FUNCTION_BLOCK FB_TwoAxisPopIn
VAR_INPUT
	RepRate : BOOL;
	
	Axis1_InsertedPos2_IN : BOOL;
	Axis1_RetractedPos1_IN : BOOL;
	
	Axis2_InsertedPos2_IN : BOOL;
	Axis2_RetractedPos1_IN : BOOL;
END_VAR
VAR_OUTPUT
	Interlock : BOOL;
	Axis1_State : E_2PosMonState;
	Axis2_State : E_2PosMonState;
	
	Axis1_InsertPos2_OUT : BOOL;
	Axis2_InsertPos2_OUT : BOOL;
END_VAR
VAR
	Axis1 : FB_TwoPositionPopIn;
	Axis2 : FB_TwoPositionPopIn;
END_VAR

// Instances of 2 and 3 position monitor
Axis1(RepRate := RepRate, 	
			Inserted_Pos2_IN := Axis1_InsertedPos2_IN,	
			Retracted_Pos1_IN := Axis1_RetractedPos1_IN,
			Insert_Pos2_OUT => Axis1_InsertPos2_OUT,
			State => Axis1_State );
			
Axis2(RepRate := RepRate,  
		Inserted_Pos2_IN := Axis2_InsertedPos2_IN, 	
		Retracted_Pos1_IN := Axis2_RetractedPos1_IN,
		Insert_Pos2_OUT => Axis2_InsertPos2_OUT, 
		State => Axis2_State);

//Handle Horizontal -  RET Air solenoid - three way position monitor collisions

IF Axis1.State = E_2PosMonState.isBROKEN AND Axis2.State= E_2PosMonState.isINSERTED THEN 
	Axis1.Retract();
ELSIF Axis1.State = E_2PosMonState.isRETRACTED AND Axis2.State = E_2PosMonState.isBROKEN THEN 
	Axis1.Retract();
ELSIF Axis1.State = E_2PosMonState.isRETRACTED AND Axis2.State = E_2PosMonState.isINSERTED THEN 
	Axis1.Retract();
ELSIF Axis1.State = E_2PosMonState.isRETRACTED AND Axis2.State = E_2PosMonState.isMOVING THEN 
	Axis1.Retract();
ELSIF Axis1.State = E_2PosMonState.isMOVING AND Axis2.State = E_2PosMonState.isINSERTED THEN 
	Axis1.Retract();
ELSIF Axis1.State = E_2PosMonState.isMOVING AND Axis2.State = E_2PosMonState.isBROKEN THEN 
	Axis1.Retract();
END_IF
			
//Handle vertical 		two way position monitor collisions	
IF Axis1.State = E_2PosMonState.isBROKEN AND Axis2.State = E_2PosMonState.isRETRACTED THEN 
	Axis2.Retract();
ELSIF Axis1.State = E_2PosMonState.isBROKEN AND Axis2.State = E_2PosMonState.isMOVING THEN 
	Axis2.Retract();
ELSIF Axis1.State = E_2PosMonState.isINSERTED AND Axis2.State = E_2PosMonState.isBROKEN THEN 
	Axis2.Retract();
ELSIF Axis1.State = E_2PosMonState.isINSERTED AND Axis2.State = E_2PosMonState.isRETRACTED THEN 
	Axis2.Retract();
ELSIF Axis1.State = E_2PosMonState.isINSERTED AND Axis2.State = E_2PosMonState.isMOVING THEN 
	Axis2.Retract();
ELSIF Axis1.State = E_2PosMonState.isMOVING AND Axis2.State = E_2PosMonState.isRETRACTED THEN 
	Axis2.Retract();
END_IF

// Handle MPS shutter Interlock output
Interlock := Axis2.Interlock AND Axis1.Interlock AND 
			(Axis1.State = E_2PosMonState.isRETRACTED AND Axis2.State = E_2PosMonState.isINSERTED) OR
			(Axis1.State = E_2PosMonState.isRETRACTED AND Axis2.State = E_2PosMonState.isRETRACTED) OR
			(Axis1.State = E_2PosMonState.isINSERTED AND Axis2.State= E_2PosMonState.isRETRACTED);

METHOD Control : BOOL
VAR_IN_OUT
	structure : ST_TwoAxisPopIn;
END_VAR
//Commands
IF structure.Axis1_InsertPos2Cmd THEN
	structure.Axis1_InsertPos2Cmd:=FALSE;
	InsertAxis1();
END_IF

IF structure.Axis1_RetractPos1Cmd THEN
	structure.Axis1_RetractPos1Cmd:=FALSE;
	RetractAxis1();
END_IF

IF structure.Axis2_InsertPos2Cmd THEN
	structure.Axis2_InsertPos2Cmd:=FALSE;
	InsertAxis2();
END_IF

IF structure.Axis2_RetractPos1Cmd THEN
	structure.Axis2_RetractPos1Cmd:=FALSE;
	RetractAxis2();
END_IF

//Statuses

structure.Axis1_IsInsertedPos2St:=Axis1.Inserted_Pos2_IN;
structure.Axis1_IsRetractedPos1St:=Axis1.Retracted_Pos1_IN;

structure.Axis2_IsInsertedPos2St:=Axis2.Inserted_Pos2_IN;
structure.Axis2_IsRetractedPos1St:=Axis2.Retracted_Pos1_IN;

structure.InterlockSt:=Interlock;

structure.Axis1StateSt:=Axis1_State;
structure.Axis2StateSt:=Axis2_State;
END_METHOD

METHOD InsertAxis1 : BOOL
VAR_INPUT
END_VAR
IF Axis1.State = E_3PosMonState.isBROKEN AND Axis2.State= E_2PosMonState.isINSERTED THEN 
	RETURN;
ELSIF Axis1.State = E_3PosMonState.isRETRACTED AND Axis2.State = E_2PosMonState.isBROKEN THEN 
	RETURN;
ELSIF Axis1.State = E_3PosMonState.isRETRACTED AND Axis2.State = E_2PosMonState.isINSERTED THEN 
	RETURN;
ELSIF Axis1.State = E_3PosMonState.isRETRACTED AND Axis2.State = E_2PosMonState.isMOVING THEN 
	RETURN;
ELSIF Axis1.State = E_3PosMonState.isMOVING AND Axis2.State = E_2PosMonState.isINSERTED THEN 
	RETURN;
ELSIF Axis1.State = E_3PosMonState.isMOVING AND Axis2.State = E_2PosMonState.isBROKEN THEN 
	RETURN;
END_IF

Axis1.Insert();
END_METHOD

METHOD InsertAxis2 : BOOL
VAR_INPUT
END_VAR
IF Axis1.State = E_2PosMonState.isBROKEN AND Axis2.State= E_2PosMonState.isRETRACTED THEN 
	RETURN;
ELSIF Axis1.State = E_2PosMonState.isBROKEN AND Axis2.State= E_2PosMonState.isMOVING THEN 
	RETURN;
ELSIF Axis1.State = E_2PosMonState.isINSERTED AND Axis2.State = E_2PosMonState.isBROKEN THEN 
	RETURN;
ELSIF Axis1.State = E_2PosMonState.isINSERTED AND Axis2.State = E_2PosMonState.isRETRACTED THEN 
	RETURN;
ELSIF Axis1.State = E_2PosMonState.isINSERTED AND Axis2.State = E_2PosMonState.isMOVING THEN 
	RETURN;
ELSIF Axis1.State = E_3PosMonState.isMOVING AND Axis2.State = E_2PosMonState.isRETRACTED THEN 
	RETURN;
END_IF

Axis2.Insert();
END_METHOD

METHOD RetractAxis1 : BOOL
VAR_INPUT
END_VAR
Axis1.Retract();
END_METHOD

METHOD RetractAxis2 : BOOL
VAR_INPUT
END_VAR
Axis2.Retract();
END_METHOD

END_FUNCTION_BLOCK

(* stored: Version 1.1.0.1, ProductVersion 3.1.4024.12
   POU FB_TwoAxisPopIn: Id {d9ee7f31-afa1-410b-aa2b-f47d1398c395}, SpecialFunc None
   Method Control: Id {1f5ffb39-0a2a-4919-bac2-be91234102e9}
   Method InsertAxis1: Id {5f8f7f28-7413-462b-8c88-d0be6ceee2d9}
   Method InsertAxis2: Id {b39fcb84-0e40-4b23-b1a7-c6b365f7c82c}
   Method RetractAxis1: Id {4a8e9af8-f62b-4608-ba07-70548710f69d}
   Method RetractAxis2: Id {7248571d-9ddf-49b7-8d83-635fd627b605} *)
